{attribute 'linkalways'} 
{attribute 'no_explicit_call' := 'This FB is a CLASS and must be accessed using methods or properties'}
{attribute 'enable_dynamic_creation'}
FUNCTION_BLOCK FINAL DIV_INT EXTENDS Node
VAR
	in1 : _INT(0);
	in2 : _INT(0);
	out : _INT(0);
	div0 : _BOOL(FALSE);
END_VAR

METHOD PUBLIC Clone : I_Node
VAR
	pNode : POINTER TO DIV_INT;
END_VAR
pNode := __NEW(DIV_INT);
Clone := pNode^;
END_METHOD

METHOD FB_init : BOOL
VAR_INPUT
	bInitRetains : BOOL; // if TRUE, the retain variables are initialized (warm start / cold start)
	bInCopyCode : BOOL;  // if TRUE, the instance afterwards gets moved into the copy code (online change)
END_VAR
AddInput('in1',THIS^.in1);
AddInput('in2',THIS^.in2);
AddOutput('out', THIS^.out);
AddOutput('div0', THIS^.div0);
END_METHOD

METHOD PROTECTED OnExecute
VAR
END_VAR
IF in2.Value = 0 THEN
	div0.Value := TRUE;
	RETURN;
END_IF

out.Value := in1.Value / in2.Value;
div0.Value := FALSE;
END_METHOD

END_FUNCTION_BLOCK

(* stored: Version 1.1.0.1, ProductVersion 3.1.4024.15
   POU DIV_INT: Id {5a194c9e-e1ec-4483-b8b5-46a33fbae3a8}, SpecialFunc None
   Folder Constructor: Id {9a2b2db5-1dd1-4227-9e45-728924e7be2e}
   Method Clone: Id {e887faed-8c4d-4214-a425-1dfc75a5f649}
   Method FB_init: Id {41b8a704-ed17-4722-9fe1-c7a55919079b}
   Method OnExecute: Id {e62557e9-8402-4f4d-8a0c-1d51d42d3383} *)
